FUNCTION_BLOCK OR_WORD (* IEC 61131-3 Bitwise OR *)
  (* Standard: 61131-3 *)
  (* Version 0.1, 2006-09-08, JHC, Holobloc Inc, Converted to Template. *)
  (* Version 0.0, 2004-12-15, JHC, Rockwell Automation, Converted from SRC format. *)
  (* Compiler header: package fb.rt.plc.bits; *)
  (* Compiler classdef: (IN1 | IN2) *)
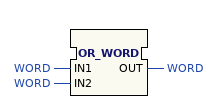
  VAR_INPUT
    IN1 : WORD;
    IN2 : WORD;
  END_VAR
  VAR_OUTPUT
    OUT : WORD;
  END_VAR
END_FUNCTION_BLOCK
